VAR_GLOBAL 
HARD:Hard;
	

END_VAR

(* stored: Version 1.1.0.1, ProductVersion 3.1.4024.9
   GVL _Hard: Id {a0de562e-a1a9-4240-92d7-3259a889751a} *)
